// TIA Portal V17 export
// export: Created 2023-04-05T06:28:00.5446237Z, ExportSetting None, DisplayName Totally Integrated Automation Portal, DisplayVersion V17 Update 4, DisplayName TIA Portal Openness, DisplayVersion V17 Update 4, DisplayName TIA Portal Version Control Interface, DisplayVersion V17, DisplayName STEP 7 Professional, DisplayVersion V17 Update 4, DisplayName STEP 7 Safety, DisplayVersion V17, DisplayName WinCC Advanced / Unified PC, DisplayVersion V17 Update 4
DATA_BLOCK "UP"   // DB51
{ S7_Optimized_Access := 'FALSE' }
// stored: AutoNumber false
   VAR RETAIN
      CMN_ALM : Bool;   // True = Alarm active
      CMN_SH : Bool;   // True = Shutdown active
      CMN_EM : Bool;   // True = Emergency active
      CMN_MOS : Bool;   // True = Mos active
      SPARE : Bool;
      SPARE2 : Bool;
      SPARE3 : Bool;
      SPARE4 : Bool;
      SPARE5 : Byte;   // Reserved for HMI ACK
      ALM_FLASHING : Int;   // Variable for alarm flashing
      TRIP_FLASHING : Int;   // Variable for trip flashing
   END_VAR
BEGIN
END_DATA_BLOCK
